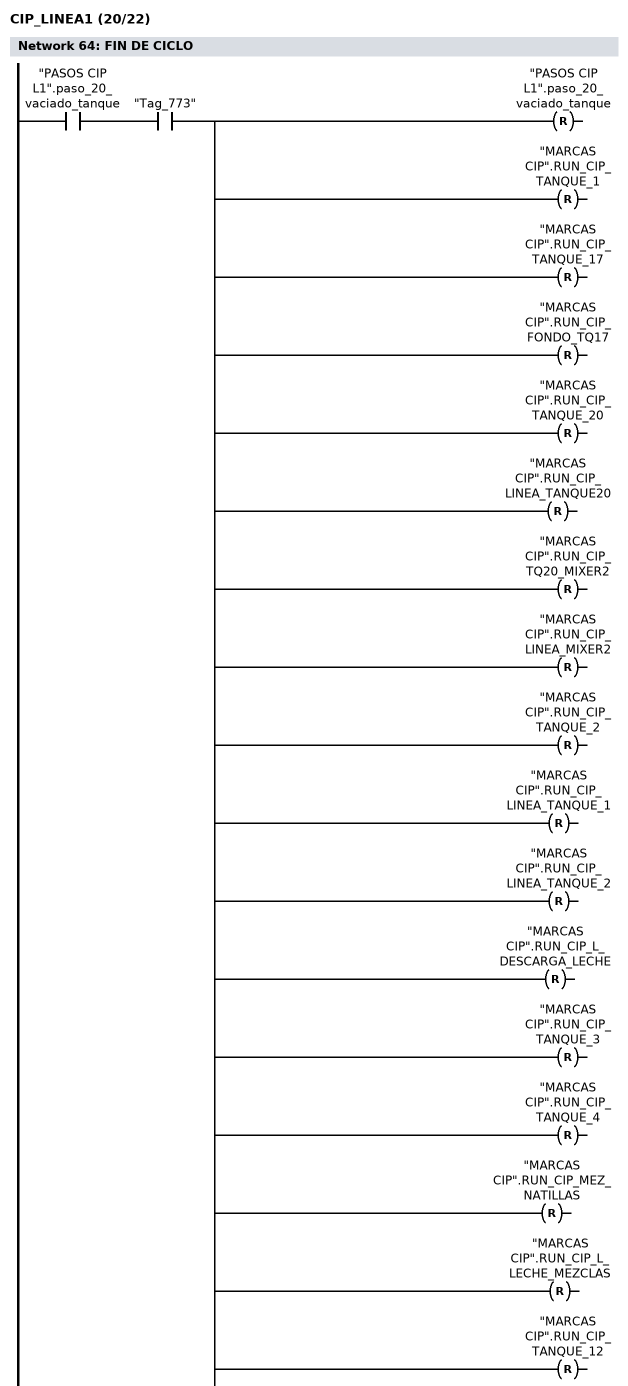
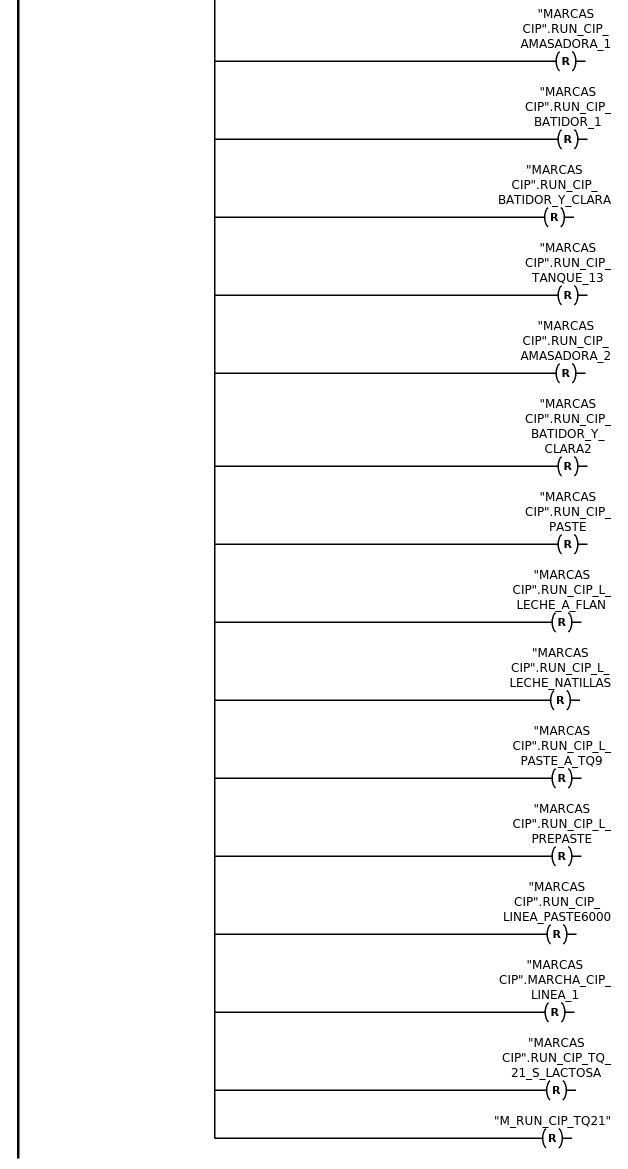
   RUNG wire#powerrail
      Contact( "PASOS CIP L1".paso_20_vaciado_tanque )
      Contact( "Tag_773" )
      wire#w1
      R_Coil( "PASOS CIP L1".paso_20_vaciado_tanque )
   END_RUNG
   RUNG wire#w1
      R_Coil( "MARCAS CIP".RUN_CIP_TANQUE_1 )
   END_RUNG
   RUNG wire#w1
      R_Coil( "MARCAS CIP".RUN_CIP_TANQUE_17 )
   END_RUNG
   RUNG wire#w1
      R_Coil( "MARCAS CIP".RUN_CIP_FONDO_TQ17 )
   END_RUNG
   RUNG wire#w1
      R_Coil( "MARCAS CIP".RUN_CIP_TANQUE_20 )
   END_RUNG
   RUNG wire#w1
      R_Coil( "MARCAS CIP".RUN_CIP_LINEA_TANQUE20 )
   END_RUNG
   RUNG wire#w1
      R_Coil( "MARCAS CIP".RUN_CIP_TQ20_MIXER2 )
   END_RUNG
   RUNG wire#w1
      R_Coil( "MARCAS CIP".RUN_CIP_LINEA_MIXER2 )
   END_RUNG
   RUNG wire#w1
      R_Coil( "MARCAS CIP".RUN_CIP_TANQUE_2 )
   END_RUNG
   RUNG wire#w1
      R_Coil( "MARCAS CIP".RUN_CIP_LINEA_TANQUE_1 )
   END_RUNG
   RUNG wire#w1
      R_Coil( "MARCAS CIP".RUN_CIP_LINEA_TANQUE_2 )
   END_RUNG
   RUNG wire#w1
      R_Coil( "MARCAS CIP".RUN_CIP_L_DESCARGA_LECHE )
   END_RUNG
   RUNG wire#w1
      R_Coil( "MARCAS CIP".RUN_CIP_TANQUE_3 )
   END_RUNG
   RUNG wire#w1
      R_Coil( "MARCAS CIP".RUN_CIP_TANQUE_4 )
   END_RUNG
   RUNG wire#w1
      R_Coil( "MARCAS CIP".RUN_CIP_MEZ_NATILLAS )
   END_RUNG
   RUNG wire#w1
      R_Coil( "MARCAS CIP".RUN_CIP_L_LECHE_MEZCLAS )
   END_RUNG
   RUNG wire#w1
      R_Coil( "MARCAS CIP".RUN_CIP_TANQUE_12 )
   END_RUNG
   RUNG wire#w1
      R_Coil( "MARCAS CIP".RUN_CIP_AMASADORA_1 )
   END_RUNG
   RUNG wire#w1
      R_Coil( "MARCAS CIP".RUN_CIP_BATIDOR_1 )
   END_RUNG
   RUNG wire#w1
      R_Coil( "MARCAS CIP".RUN_CIP_BATIDOR_Y_CLARA )
   END_RUNG
   RUNG wire#w1
      R_Coil( "MARCAS CIP".RUN_CIP_TANQUE_13 )
   END_RUNG
   RUNG wire#w1
      R_Coil( "MARCAS CIP".RUN_CIP_AMASADORA_2 )
   END_RUNG
   RUNG wire#w1
      R_Coil( "MARCAS CIP".RUN_CIP_BATIDOR_Y_CLARA2 )
   END_RUNG
   RUNG wire#w1
      R_Coil( "MARCAS CIP".RUN_CIP_PASTE )
   END_RUNG
   RUNG wire#w1
      R_Coil( "MARCAS CIP".RUN_CIP_L_LECHE_A_FLAN )
   END_RUNG
   RUNG wire#w1
      R_Coil( "MARCAS CIP".RUN_CIP_L_LECHE_NATILLAS )
   END_RUNG
   RUNG wire#w1
      R_Coil( "MARCAS CIP".RUN_CIP_L_PASTE_A_TQ9 )
   END_RUNG
   RUNG wire#w1
      R_Coil( "MARCAS CIP".RUN_CIP_L_PREPASTE )
   END_RUNG
   RUNG wire#w1
      R_Coil( "MARCAS CIP".RUN_CIP_LINEA_PASTE6000 )
   END_RUNG
   RUNG wire#w1
      R_Coil( "MARCAS CIP".MARCHA_CIP_LINEA_1 )
   END_RUNG
   RUNG wire#w1
      R_Coil( "MARCAS CIP".RUN_CIP_TQ_21_S_LACTOSA )
   END_RUNG
   RUNG wire#w1
      R_Coil( "M_RUN_CIP_TQ21" )
   END_RUNG
   // the same network as SCL:
   #_w1 := "PASOS CIP L1".paso_20_vaciado_tanque AND "Tag_773";
   IF #_w1 THEN
       "PASOS CIP L1".paso_20_vaciado_tanque := FALSE;
       "MARCAS CIP".RUN_CIP_TANQUE_1 := FALSE;
       "MARCAS CIP".RUN_CIP_TANQUE_17 := FALSE;
       "MARCAS CIP".RUN_CIP_FONDO_TQ17 := FALSE;
       "MARCAS CIP".RUN_CIP_TANQUE_20 := FALSE;
       "MARCAS CIP".RUN_CIP_LINEA_TANQUE20 := FALSE;
       "MARCAS CIP".RUN_CIP_TQ20_MIXER2 := FALSE;
       "MARCAS CIP".RUN_CIP_LINEA_MIXER2 := FALSE;
       "MARCAS CIP".RUN_CIP_TANQUE_2 := FALSE;
       "MARCAS CIP".RUN_CIP_LINEA_TANQUE_1 := FALSE;
       "MARCAS CIP".RUN_CIP_LINEA_TANQUE_2 := FALSE;
       "MARCAS CIP".RUN_CIP_L_DESCARGA_LECHE := FALSE;
       "MARCAS CIP".RUN_CIP_TANQUE_3 := FALSE;
       "MARCAS CIP".RUN_CIP_TANQUE_4 := FALSE;
       "MARCAS CIP".RUN_CIP_MEZ_NATILLAS := FALSE;
       "MARCAS CIP".RUN_CIP_L_LECHE_MEZCLAS := FALSE;
       "MARCAS CIP".RUN_CIP_TANQUE_12 := FALSE;
       "MARCAS CIP".RUN_CIP_AMASADORA_1 := FALSE;
       "MARCAS CIP".RUN_CIP_BATIDOR_1 := FALSE;
       "MARCAS CIP".RUN_CIP_BATIDOR_Y_CLARA := FALSE;
       "MARCAS CIP".RUN_CIP_TANQUE_13 := FALSE;
       "MARCAS CIP".RUN_CIP_AMASADORA_2 := FALSE;
       "MARCAS CIP".RUN_CIP_BATIDOR_Y_CLARA2 := FALSE;
       "MARCAS CIP".RUN_CIP_PASTE := FALSE;
       "MARCAS CIP".RUN_CIP_L_LECHE_A_FLAN := FALSE;
       "MARCAS CIP".RUN_CIP_L_LECHE_NATILLAS := FALSE;
       "MARCAS CIP".RUN_CIP_L_PASTE_A_TQ9 := FALSE;
       "MARCAS CIP".RUN_CIP_L_PREPASTE := FALSE;
       "MARCAS CIP".RUN_CIP_LINEA_PASTE6000 := FALSE;
       "MARCAS CIP".MARCHA_CIP_LINEA_1 := FALSE;
       "MARCAS CIP".RUN_CIP_TQ_21_S_LACTOSA := FALSE;
       "M_RUN_CIP_TQ21" := FALSE;
   END_IF;
END_REGION

REGION Network 65: Variable prvisional
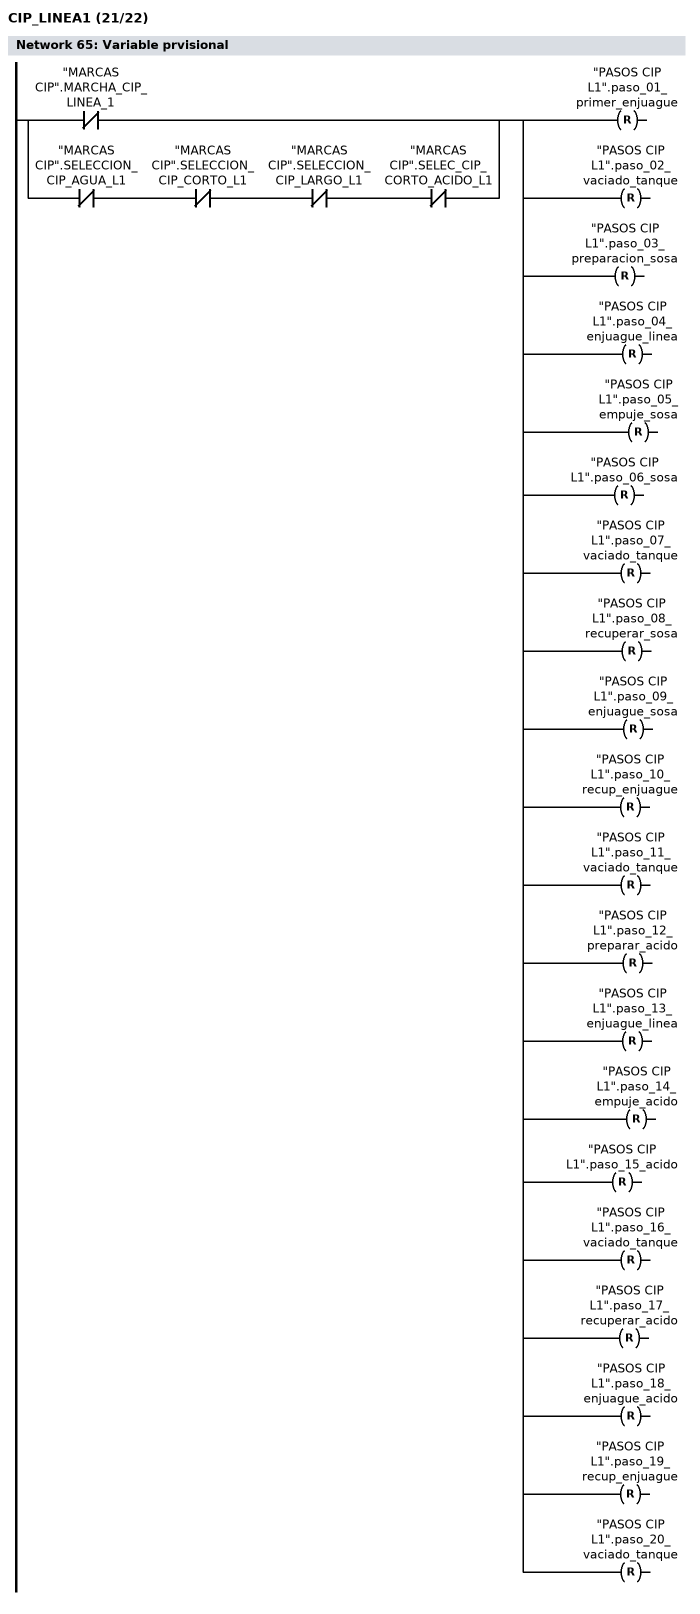
   RUNG wire#powerrail
      I_Contact( "MARCAS CIP".MARCHA_CIP_LINEA_1 )
      wire#w1
      R_Coil( "PASOS CIP L1".paso_01_primer_enjuague )
   END_RUNG
   RUNG wire#powerrail
      I_Contact( "MARCAS CIP".SELECCION_CIP_AGUA_L1 )
      I_Contact( "MARCAS CIP".SELECCION_CIP_CORTO_L1 )
      I_Contact( "MARCAS CIP".SELECCION_CIP_LARGO_L1 )
      I_Contact( "MARCAS CIP".SELEC_CIP_CORTO_ACIDO_L1 )
   END_RUNG wire#w1
   RUNG wire#w1
      R_Coil( "PASOS CIP L1".paso_02_vaciado_tanque )
   END_RUNG
   RUNG wire#w1
      R_Coil( "PASOS CIP L1".paso_03_preparacion_sosa )
   END_RUNG
   RUNG wire#w1
      R_Coil( "PASOS CIP L1".paso_04_enjuague_linea )
   END_RUNG
   RUNG wire#w1
      R_Coil( "PASOS CIP L1".paso_05_empuje_sosa )
   END_RUNG
   RUNG wire#w1
      R_Coil( "PASOS CIP L1".paso_06_sosa )
   END_RUNG
   RUNG wire#w1
      R_Coil( "PASOS CIP L1".paso_07_vaciado_tanque )
   END_RUNG
   RUNG wire#w1
      R_Coil( "PASOS CIP L1".paso_08_recuperar_sosa )
   END_RUNG
   RUNG wire#w1
      R_Coil( "PASOS CIP L1".paso_09_enjuague_sosa )
   END_RUNG
   RUNG wire#w1
      R_Coil( "PASOS CIP L1".paso_10_recup_enjuague )
   END_RUNG
   RUNG wire#w1
      R_Coil( "PASOS CIP L1".paso_11_vaciado_tanque )
   END_RUNG
   RUNG wire#w1
      R_Coil( "PASOS CIP L1".paso_12_preparar_acido )
   END_RUNG
   RUNG wire#w1
      R_Coil( "PASOS CIP L1".paso_13_enjuague_linea )
   END_RUNG
   RUNG wire#w1
      R_Coil( "PASOS CIP L1".paso_14_empuje_acido )
   END_RUNG
   RUNG wire#w1
      R_Coil( "PASOS CIP L1".paso_15_acido )
   END_RUNG
   RUNG wire#w1
      R_Coil( "PASOS CIP L1".paso_16_vaciado_tanque )
   END_RUNG
   RUNG wire#w1
      R_Coil( "PASOS CIP L1".paso_17_recuperar_acido )
   END_RUNG
   RUNG wire#w1
      R_Coil( "PASOS CIP L1".paso_18_enjuague_acido )
   END_RUNG
   RUNG wire#w1
      R_Coil( "PASOS CIP L1".paso_19_recup_enjuague )
   END_RUNG
   RUNG wire#w1
      R_Coil( "PASOS CIP L1".paso_20_vaciado_tanque )
   END_RUNG
   // the same network as SCL:
   IF NOT "MARCAS CIP".MARCHA_CIP_LINEA_1 OR (NOT "MARCAS CIP".SELECCION_CIP_AGUA_L1 AND NOT "MARCAS CIP".SELECCION_CIP_CORTO_L1 AND NOT "MARCAS CIP".SELECCION_CIP_LARGO_L1 AND NOT "MARCAS CIP".SELEC_CIP_CORTO_ACIDO_L1) THEN
       "PASOS CIP L1".paso_01_primer_enjuague := FALSE;
       "PASOS CIP L1".paso_02_vaciado_tanque := FALSE;
       "PASOS CIP L1".paso_03_preparacion_sosa := FALSE;
       "PASOS CIP L1".paso_04_enjuague_linea := FALSE;
       "PASOS CIP L1".paso_05_empuje_sosa := FALSE;
       "PASOS CIP L1".paso_06_sosa := FALSE;
       "PASOS CIP L1".paso_07_vaciado_tanque := FALSE;
       "PASOS CIP L1".paso_08_recuperar_sosa := FALSE;
       "PASOS CIP L1".paso_09_enjuague_sosa := FALSE;
       "PASOS CIP L1".paso_10_recup_enjuague := FALSE;
       "PASOS CIP L1".paso_11_vaciado_tanque := FALSE;
       "PASOS CIP L1".paso_12_preparar_acido := FALSE;
       "PASOS CIP L1".paso_13_enjuague_linea := FALSE;
       "PASOS CIP L1".paso_14_empuje_acido := FALSE;
       "PASOS CIP L1".paso_15_acido := FALSE;
       "PASOS CIP L1".paso_16_vaciado_tanque := FALSE;
       "PASOS CIP L1".paso_17_recuperar_acido := FALSE;
       "PASOS CIP L1".paso_18_enjuague_acido := FALSE;
       "PASOS CIP L1".paso_19_recup_enjuague := FALSE;
       "PASOS CIP L1".paso_20_vaciado_tanque := FALSE;
   END_IF;
END_REGION

REGION Network 66
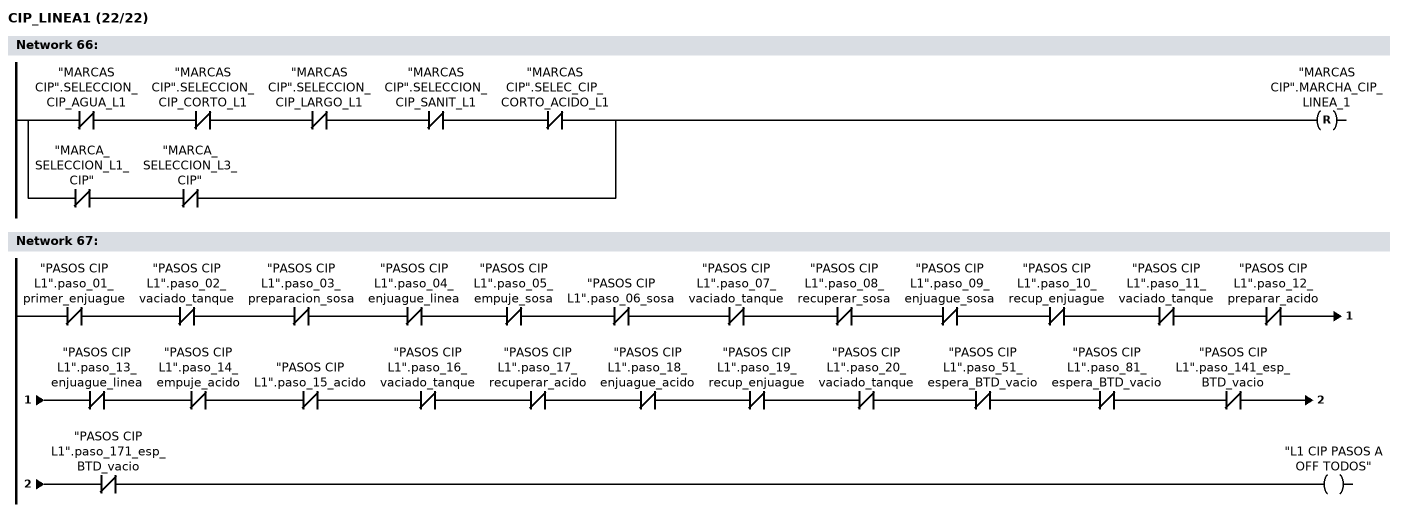
   RUNG wire#powerrail
      I_Contact( "MARCAS CIP".SELECCION_CIP_AGUA_L1 )
      I_Contact( "MARCAS CIP".SELECCION_CIP_CORTO_L1 )
      I_Contact( "MARCAS CIP".SELECCION_CIP_LARGO_L1 )
      I_Contact( "MARCAS CIP".SELECCION_CIP_SANIT_L1 )
      I_Contact( "MARCAS CIP".SELEC_CIP_CORTO_ACIDO_L1 )
      wire#w1
      R_Coil( "MARCAS CIP".MARCHA_CIP_LINEA_1 )
   END_RUNG
   RUNG wire#powerrail
      I_Contact( "MARCA_SELECCION_L1_CIP" )
      I_Contact( "MARCA_SELECCION_L3_CIP" )
   END_RUNG wire#w1
   // the same network as SCL:
   IF (NOT "MARCAS CIP".SELECCION_CIP_AGUA_L1 AND NOT "MARCAS CIP".SELECCION_CIP_CORTO_L1 AND NOT "MARCAS CIP".SELECCION_CIP_LARGO_L1 AND NOT "MARCAS CIP".SELECCION_CIP_SANIT_L1 AND NOT "MARCAS CIP".SELEC_CIP_CORTO_ACIDO_L1) OR (NOT "MARCA_SELECCION_L1_CIP" AND NOT "MARCA_SELECCION_L3_CIP") THEN
       "MARCAS CIP".MARCHA_CIP_LINEA_1 := FALSE;
   END_IF;
END_REGION

REGION Network 67
   RUNG wire#powerrail
      I_Contact( "PASOS CIP L1".paso_01_primer_enjuague )
      I_Contact( "PASOS CIP L1".paso_02_vaciado_tanque )
      I_Contact( "PASOS CIP L1".paso_03_preparacion_sosa )
      I_Contact( "PASOS CIP L1".paso_04_enjuague_linea )
      I_Contact( "PASOS CIP L1".paso_05_empuje_sosa )
      I_Contact( "PASOS CIP L1".paso_06_sosa )
      I_Contact( "PASOS CIP L1".paso_07_vaciado_tanque )
      I_Contact( "PASOS CIP L1".paso_08_recuperar_sosa )
      I_Contact( "PASOS CIP L1".paso_09_enjuague_sosa )
      I_Contact( "PASOS CIP L1".paso_10_recup_enjuague )
      I_Contact( "PASOS CIP L1".paso_11_vaciado_tanque )
      I_Contact( "PASOS CIP L1".paso_12_preparar_acido )
      I_Contact( "PASOS CIP L1".paso_13_enjuague_linea )
      I_Contact( "PASOS CIP L1".paso_14_empuje_acido )
      I_Contact( "PASOS CIP L1".paso_15_acido )
      I_Contact( "PASOS CIP L1".paso_16_vaciado_tanque )
      I_Contact( "PASOS CIP L1".paso_17_recuperar_acido )
      I_Contact( "PASOS CIP L1".paso_18_enjuague_acido )
      I_Contact( "PASOS CIP L1".paso_19_recup_enjuague )
      I_Contact( "PASOS CIP L1".paso_20_vaciado_tanque )
      I_Contact( "PASOS CIP L1".paso_51_espera_BTD_vacio )
      I_Contact( "PASOS CIP L1".paso_81_espera_BTD_vacio )
      I_Contact( "PASOS CIP L1".paso_141_esp_BTD_vacio )
      I_Contact( "PASOS CIP L1".paso_171_esp_BTD_vacio )
      Coil( "L1 CIP PASOS A OFF TODOS" )
   END_RUNG
   // the same network as SCL:
   "L1 CIP PASOS A OFF TODOS" := NOT "PASOS CIP L1".paso_01_primer_enjuague AND NOT "PASOS CIP L1".paso_02_vaciado_tanque AND NOT "PASOS CIP L1".paso_03_preparacion_sosa AND NOT "PASOS CIP L1".paso_04_enjuague_linea AND NOT "PASOS CIP L1".paso_05_empuje_sosa AND NOT "PASOS CIP L1".paso_06_sosa AND NOT "PASOS CIP L1".paso_07_vaciado_tanque AND NOT "PASOS CIP L1".paso_08_recuperar_sosa AND NOT "PASOS CIP L1".paso_09_enjuague_sosa AND NOT "PASOS CIP L1".paso_10_recup_enjuague AND NOT "PASOS CIP L1".paso_11_vaciado_tanque AND NOT "PASOS CIP L1".paso_12_preparar_acido AND NOT "PASOS CIP L1".paso_13_enjuague_linea AND NOT "PASOS CIP L1".paso_14_empuje_acido AND NOT "PASOS CIP L1".paso_15_acido AND NOT "PASOS CIP L1".paso_16_vaciado_tanque AND NOT "PASOS CIP L1".paso_17_recuperar_acido AND NOT "PASOS CIP L1".paso_18_enjuague_acido AND NOT "PASOS CIP L1".paso_19_recup_enjuague AND NOT "PASOS CIP L1".paso_20_vaciado_tanque AND NOT "PASOS CIP L1".paso_51_espera_BTD_vacio AND NOT "PASOS CIP L1".paso_81_espera_BTD_vacio AND NOT "PASOS CIP L1".paso_141_esp_BTD_vacio AND NOT "PASOS CIP L1".paso_171_esp_BTD_vacio;
END_REGION
END_FUNCTION
